ABB RobotStudio station: Tp2_20201211-190708.rsstn

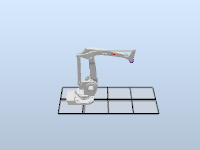
Station Solution5 (saved by RobotStudio 20.1.8982.0)
Layout (positions relative to the parent item):
  - IRB660_180_315__01 [mechanism, from Robots\IRB660_180_315__01.rslib] at (0, 0, 0) mm; joint values [0, 0, 0, 0] (rad or m)
